INTERFACE I_MotionAxisDS402NC  EXTENDS I_MotionAxisCommon

(*
    Check all post condition before updating bCommandedMoveAbsolute
    The implmentatation will depend on the axis type
    DS402 NC/Direct axis : Implementation need to check that the drive is in the correct mode before initaiting the move then set bCommandedMoveAbsolute
    MP NC axis : will immediately write to bCommandedMoveAbsolute
*)
METHOD StartMove : BOOL
VAR_INPUT
	MoveMode	: E_EpicsMotorCmd;
	CmdExecute	: BOOL;
END_VAR
END_METHOD

END_INTERFACE

(* stored: Version 1.1.0.1
   Itf I_MotionAxisDS402NC: Id {245da5fa-2b8b-4997-8294-23517a0558b2}
   Method StartMove: Id {08a6e43a-3d73-4123-9713-aea8773a1f67} *)
